// LS Electric XG5000 project: 동남91_1
// PLC NewPLC
// module base 0 slot 0: 입출력 모듈:XBC-DN/DP14E (DC 24V 입력 8점, 트랜지스터 출력 6점)

PROGRAM NewProgram (task: 스캔 프로그램)

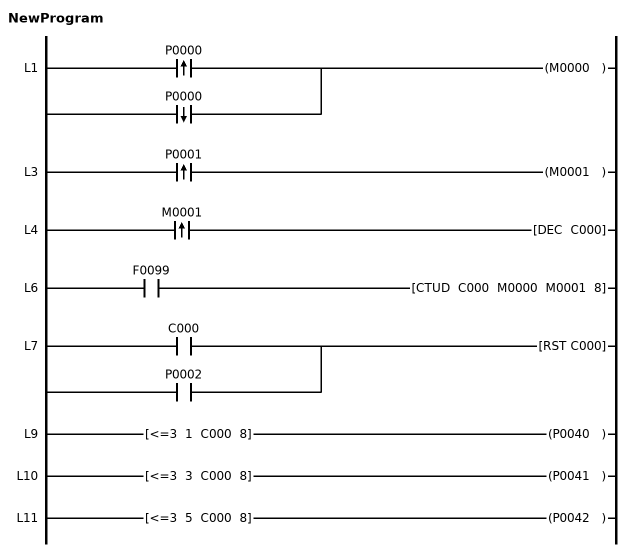
; L1
LOADP     P0000
ORN       P0000
OUT       M0000
; L3
LOADP     P0001
OUT       M0001
; L4
LOADP     M0001
DEC       C000
; L6
LOAD      F0099
CTUD      C000 M0000 M0001 8
; L7
LOAD      C000
OR        P0002
RST       C000
; L9
LOAD<=3   1 C000 8
OUT       P0040
; L10
LOAD<=3   3 C000 8
OUT       P0041
; L11
LOAD<=3   5 C000 8
OUT       P0042